FUNCTION_BLOCK Time_Out_Actuator_CommandAndMoved2 (* Basic FB with empty ECC *)
  (* Standard: 61499-2 *)
  (* Version 1.0, 2023-03-16, AK125171 *)
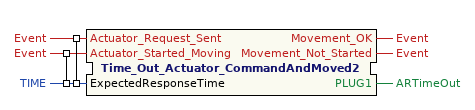
  EVENT_INPUT
    Actuator_Request_Sent WITH ExpectedResponseTime;
    Actuator_Started_Moving WITH ExpectedResponseTime;
  END_EVENT
  EVENT_OUTPUT
    Movement_OK;
    Movement_Not_Started;
  END_EVENT
  VAR_INPUT
    ExpectedResponseTime : TIME;
  END_VAR
  PLUGS
    PLUG1 : ARTimeOut;
  END_PLUGS
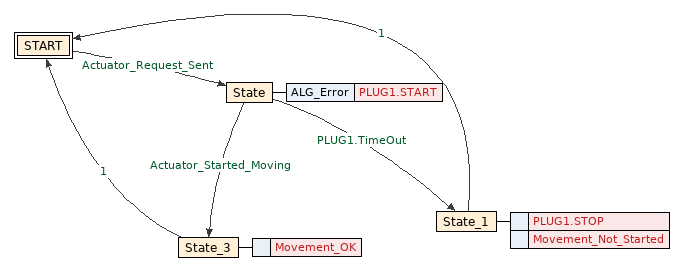
  EC_STATES
    START; (* Initial State *)
    State : ALG_Error -> PLUG1.START;
    State_3 : -> Movement_OK;
    State_1 : -> PLUG1.STOP, -> Movement_Not_Started;
  END_STATES
  EC_TRANSITIONS
    START TO State := Actuator_Request_Sent;
    State_3 TO START := 1;
    State TO State_1 := PLUG1.TimeOut;
    State_1 TO START := 1;
    State TO State_3 := Actuator_Started_Moving;
  END_TRANSITIONS
  ALGORITHM ALG_Error IN ST:
Plug1.DT:=ExpectedResponseTime;
  END_ALGORITHM
END_FUNCTION_BLOCK
